// TwinCAT 3 PLC project PlcProject
// ProgramVersion: 3.1.4023.0
// libraries:
//   lcls-twincat-motion, * (SLAC)
//   Tc2_EtherCAT, * (Beckhoff Automation GmbH)
//   Tc2_IoFunctions, * (Beckhoff Automation GmbH)
//   Tc2_MC2, * (Beckhoff Automation GmbH)
//   Tc2_Standard, * (Beckhoff Automation GmbH)
//   Tc2_System, * (Beckhoff Automation GmbH)
//   Tc2_Utilities, * (Beckhoff Automation GmbH)
//   Tc3_Module, * (Beckhoff Automation GmbH)
// project tree:
//   / PlcTask.TcTTO
//   POUs/ MAIN.TcPOU, PRG_VLS_MOTION.TcPOU
// real-time tasks:
//   TASK PlcTask: cycle T#10ms, priority 20, ADS port 350
// motion (NC):
//   TASK NC-Task 1 SAF: cycle T#2ms, priority 4, ADS port 501
//   TASK NC-Task 1 SVB: cycle T#10ms, priority 8, ADS port 511
//   AXIS VLS-Slit-Right (id 1)
//     Dynamic: AccelerationMaximum=10, DecelerationMaximum=10, Acceleration=2.29041, Deceleration=2.29041, Jerk=19.7962
//     Velo: RefSearch=0.1, RefSync=0.1, SlowManual=0.5, FastManual=1, Maximum=0.5
//     OtherSettings: AllowMotionCmdToSlave=true, PulseDistancePos=1, PulseDistanceNeg=1
//     encoder EncType=4
//       EncPara: ScaleFactorNumerator=3.90625e-05, Inverse=true, MaxCount=#x0000ffff
//         SoftEndMinControl: Enable=true, Range=-48.4338
//         SoftEndMaxControl: Enable=true
//         Inc: RefSoftSyncMask=#x0000ffff
//     drive DrvType=24
//       DrvPara: Inverse=true
//         Analog: VeloReferenz=5, ScaleFactorActTorque=0.1
//         TimeComp: TaskDelayCycles=1
//     controller CtrType=2
//       CtrPara: PriorControlFactor=1
//         PosDiffControl: Range=0.1
//         PID: DeadBandPosition=0.1
//         Observer: BandWidth=20
//   AXIS VLS-Slit-Left (id 2)
//     Dynamic: AccelerationMaximum=10, DecelerationMaximum=10, Acceleration=4.49102, Deceleration=4.49102, Jerk=20.1692
//     Velo: RefSearch=0.1, RefSync=0.1, SlowManual=0.5, FastManual=1, Maximum=0.5
//     OtherSettings: AllowMotionCmdToSlave=true, PulseDistancePos=1, PulseDistanceNeg=1
//     encoder EncType=4
//       EncPara: ScaleFactorNumerator=3.90625e-05, MaxCount=#x0000ffff
//         Inc: RefSoftSyncMask=#x0000ffff
//     drive DrvType=24
//       Analog: VeloReferenz=5, ScaleFactorActTorque=0.1
//       TimeComp: TaskDelayCycles=1
//     controller CtrType=2
//       CtrPara: PriorControlFactor=1
//         PosDiffControl: Range=0.1
//         PID: DeadBandPosition=0.1
//         Observer: BandWidth=20
//   AXIS VLS-Slit-Down (id 3)
//     Dynamic: AccelerationMaximum=10, DecelerationMaximum=10, Acceleration=4.49102, Deceleration=4.49102, Jerk=20.1692
//     Velo: RefSearch=0.1, RefSync=0.1, SlowManual=0.5, FastManual=1, Maximum=1
//     OtherSettings: AllowMotionCmdToSlave=true, PulseDistancePos=1, PulseDistanceNeg=1
//     encoder EncType=4
//       EncPara: ScaleFactorNumerator=3.90625e-05, MaxCount=#x0000ffff
//         Inc: RefSoftSyncMask=#x0000ffff
//     drive DrvType=24
//       Analog: VeloReferenz=5, ScaleFactorActTorque=0.1
//       TimeComp: TaskDelayCycles=1
//     controller CtrType=2
//       CtrPara: PriorControlFactor=1
//         PosDiffControl: Range=0.1
//         PID: DeadBandPosition=0.1
//         Observer: BandWidth=20
//   AXIS VLS-Slit-Up (id 4)
//     Dynamic: AccelerationMaximum=10, DecelerationMaximum=10, Acceleration=4.49102, Deceleration=4.49102, Jerk=20.1692
//     Velo: RefSearch=0.1, RefSync=0.1, SlowManual=0.5, FastManual=1, Maximum=1
//     OtherSettings: AllowMotionCmdToSlave=true, PulseDistancePos=1, PulseDistanceNeg=1
//     encoder EncType=4
//       EncPara: ScaleFactorNumerator=3.90625e-05, MaxCount=#x0000ffff
//         Inc: RefSoftSyncMask=#x0000ffff
//     drive DrvType=24
//       Analog: VeloReferenz=5, ScaleFactorActTorque=0.1
//       TimeComp: TaskDelayCycles=1
//     controller CtrType=2
//       CtrPara: PriorControlFactor=1
//         PosDiffControl: Range=0.1
//         PID: DeadBandPosition=0.1
//         Observer: BandWidth=20
//   AXIS VLS-Focus-Mirror (id 5)
//     Dynamic: AccelerationMaximum=4, DecelerationMaximum=4, Acceleration=1.92472, Deceleration=1.92472, Jerk=18.5227
//     Velo: RefSearch=0.05, RefSync=0.05, SlowManual=0.05, FastManual=0.1, Maximum=0.4
//     OtherSettings: AllowMotionCmdToSlave=true, PulseDistancePos=0.1, PulseDistanceNeg=0.1
//     encoder EncType=4
//       EncPara: ScaleFactorNumerator=2.48046875e-05, Inverse=true, MaxCount=#x0000ffff
//         SoftEndMinControl: Enable=true
//         SoftEndMaxControl: Enable=true, Range=4.59
//         Inc: RefSoftSyncMask=#x0000ffff
//     drive DrvType=24
//       DrvPara: Inverse=true
//         Analog: VeloReferenz=3.175, ScaleFactorActTorque=0.1
//         TimeComp: TaskDelayCycles=1
//     controller CtrType=2
//       CtrPara: PriorControlFactor=1
//         PosDiffControl: Range=0.1
//         PID: DeadBandPosition=0.1
//         Observer: BandWidth=20
//   AXIS VLS-Grating (id 6)
//     Dynamic: AccelerationMaximum=10, DecelerationMaximum=10, Acceleration=4.49102, Deceleration=4.49102, Jerk=20.1692
//     Velo: RefSearch=0.1, RefSync=0.1, SlowManual=0.25, FastManual=0.5, Maximum=0.1
//     OtherSettings: AllowMotionCmdToSlave=true, PulseDistancePos=0.5, PulseDistanceNeg=0.5
//     encoder EncType=4
//       EncPara: ScaleFactorNumerator=3.90625e-06, Inverse=true, MaxCount=#x0000ffff
//         SoftEndMinControl: Enable=true
//         SoftEndMaxControl: Enable=true, Range=2.9933
//         Inc: RefSoftSyncMask=#x0000ffff
//     drive DrvType=24
//       DrvPara: Inverse=true
//         Analog: VeloReferenz=0.5, ScaleFactorActTorque=0.1
//         TimeComp: TaskDelayCycles=1
//     controller CtrType=2
//       CtrPara: PriorControlFactor=1
//         PosDiffControl: Range=0.2
//         PID: DeadBandPosition=0.1
//         Observer: BandWidth=20
//   AXIS VLS-Camera-Dist (id 7)
//     Dynamic: AccelerationMaximum=1.8, DecelerationMaximum=1.8, Acceleration=0.89, Deceleration=0.89, Jerk=3.83306
//     Velo: RefSearch=0.05, RefSync=0.05, SlowManual=0.05, FastManual=0.1, Maximum=0.4
//     OtherSettings: AllowMotionCmdToSlave=true, PulseDistancePos=1, PulseDistanceNeg=1
//     encoder EncType=4
//       EncPara: ScaleFactorNumerator=4.097617188e-06, MaxCount=#x0000ffff
//         Inc: RefSoftSyncMask=#x0000ffff
//     drive DrvType=24
//       Analog: VeloReferenz=0.524495, ScaleFactorActTorque=0.1
//       TimeComp: TaskDelayCycles=1
//     controller CtrType=2
//       CtrPara: PriorControlFactor=1
//         PosDiffControl: Range=0.1
//         PID: DeadBandPosition=0.1
//         Observer: BandWidth=20
//   AXIS VLS-Camera-Pitch (id 8)
//     General: UnitName=Degree
//     Dynamic: AccelerationMaximum=0.2, DecelerationMaximum=0.2, Acceleration=0.112494, Deceleration=0.112494, Jerk=0.506199
//     Velo: RefSearch=0.01, RefSync=0.01, SlowManual=0.01, FastManual=0.02, Maximum=0.02
//     OtherSettings: AllowMotionCmdToSlave=true, PulseDistancePos=0.1, PulseDistanceNeg=0.1
//     encoder EncType=4
//       EncPara: ScaleFactorNumerator=5.3515625e-07, Inverse=true, MaxCount=#x0000ffff
//         Inc: RefMode=2, RefSoftSyncMask=#x0000ffff
//     drive DrvType=24
//       DrvPara: Inverse=true
//         Analog: VeloReferenz=0.0685, ScaleFactorActTorque=0.1
//         TimeComp: TaskDelayCycles=1
//     controller CtrType=2
//       CtrPara: PriorControlFactor=1
//         PosDiffControl: Range=0.1
//         PID: DeadBandPosition=0.1
//         Observer: BandWidth=20
// I/O:
//   DEVICE Device 1 (EtherCAT), AmsNetId 5.65.203.216.2.1
//     Term 2 (EK1200) [EK1200-5000 EtherCAT Power supply (2A E-Bus)]
//       Term 1 (EK1122-0008) [EK1122-0008 2 port EtherCAT junction M8]
//         VLS_EP7041-3002_E1 [EP7041-3002 1Ch. Stepper motor output stage (50V, 5A)]
//         VLS_EP7041-3002_E2 [EP7041-3002 1Ch. Stepper motor output stage (50V, 5A)]
//         VLS_EP7041-3002_E3 [EP7041-3002 1Ch. Stepper motor output stage (50V, 5A)]
//         VLS_EP7041-1002_E4 [EP7041-1002 1Ch. Stepper motor output stage (50V, 1.5A)]
//         VLS_EP7041-1002_E5 [EP7041-1002 1Ch. Stepper motor output stage (50V, 1.5A)]
//         VLS_EP7041-1002_E6 [EP7041-1002 1Ch. Stepper motor output stage (50V, 1.5A)]
//         VLS_EP7041-1002_E7 [EP7041-1002 1Ch. Stepper motor output stage (50V, 1.5A)]
//         VLS_EP7041-1002_E8 [EP7041-1002 1Ch. Stepper motor output stage (50V, 1.5A)]
// variable links:
//   (this object) <-> Device 1 (EtherCAT)/Term 2 (EK1200)/Term 1 (EK1122-0008)/VLS_EP7041-3002_E1
//     Drive/Inputs/In/nState1 @bit 3 <-> STM Status/Status/Error
//     Drive/Inputs/In/nState1 @bit 7 <-> STM Status/Status/Motor stall
//     Drive/Inputs/In/nState1 @bit 5 <-> STM Status/Status/Moving negative
//     Drive/Inputs/In/nState1 @bit 4 <-> STM Status/Status/Moving positive
//     Drive/Inputs/In/nState1 @bit 1 <-> STM Status/Status/Ready
//     Drive/Inputs/In/nState1 <-> STM Status/Status/Ready to enable
//     Drive/Inputs/In/nState1 @bit 6 <-> STM Status/Status/Torque reduced
//     Drive/Inputs/In/nState1 @bit 2 <-> STM Status/Status/Warning
//     Drive/Inputs/In/nState2 @bit 3 <-> STM Status/Status/Digital input 1
//     Drive/Inputs/In/nState2 @bit 4 <-> STM Status/Status/Digital input 2
//     Drive/Inputs/In/nState2 @bit 5 <-> STM Status/Status/Sync error
//     Drive/Inputs/In/nState2 @bit 7 <-> STM Status/Status/TxPDO Toggle
//     Drive/Inputs/In/nState4 @bit 1 <-> WcState/InputToggle
//     Drive/Inputs/In/nState4 <-> WcState/WcState
//     Drive/Outputs/Out/nCtrl1 <-> STM Control/Control/Enable
//     Drive/Outputs/Out/nCtrl1 @bit 2 <-> STM Control/Control/Reduce torque
//     Drive/Outputs/Out/nCtrl1 @bit 1 <-> STM Control/Control/Reset
//     Drive/Outputs/Out/nCtrl2 @bit 3 <-> STM Control/Control/Digital output 1
//     Drive/Outputs/Out/nDataOut2[0] <-> STM Velocity/Velocity
//     Enc/Inputs/In/nDataIn1[0] <-> ENC Status compact/Counter value
//     Enc/Inputs/In/nDataIn2[0] <-> ENC Status compact/Latch value
//     Enc/Inputs/In/nState1 @bit 4 <-> ENC Status compact/Status/Counter overflow
//     Enc/Inputs/In/nState1 @bit 3 <-> ENC Status compact/Status/Counter underflow
//     Enc/Inputs/In/nState1 @bit 7 <-> ENC Status compact/Status/Extrapolation stall
//     Enc/Inputs/In/nState1 <-> ENC Status compact/Status/Latch C valid
//     Enc/Inputs/In/nState1 @bit 1 <-> ENC Status compact/Status/Latch extern valid
//     Enc/Inputs/In/nState1 @bit 2 <-> ENC Status compact/Status/Set counter done
//     Enc/Inputs/In/nState2 @bit 4 <-> ENC Status compact/Status/Status of extern latch
//     Enc/Inputs/In/nState2 <-> ENC Status compact/Status/Status of input A
//     Enc/Inputs/In/nState2 @bit 1 <-> ENC Status compact/Status/Status of input B
//     Enc/Inputs/In/nState2 @bit 2 <-> ENC Status compact/Status/Status of input C
//     Enc/Inputs/In/nState2 @bit 5 <-> ENC Status compact/Status/Sync error
//     Enc/Inputs/In/nState2 @bit 7 <-> ENC Status compact/Status/TxPDO Toggle
//     Enc/Inputs/In/nState4 @bit 1 <-> WcState/InputToggle
//     Enc/Inputs/In/nState4 <-> WcState/WcState
//     Enc/Outputs/Out/nCtrl1 <-> ENC Control compact/Control/Enable latch C
//     Enc/Outputs/Out/nCtrl1 @bit 3 <-> ENC Control compact/Control/Enable latch extern on negative edge
//     Enc/Outputs/Out/nCtrl1 @bit 1 <-> ENC Control compact/Control/Enable latch extern on positive edge
//     Enc/Outputs/Out/nCtrl1 @bit 2 <-> ENC Control compact/Control/Set counter
//     Enc/Outputs/Out/nDataOut1[0] <-> ENC Control compact/Set counter value
//   (this object) <-> Device 1 (EtherCAT)/Term 2 (EK1200)/Term 1 (EK1122-0008)/VLS_EP7041-3002_E2
//     Drive/Inputs/In/nState1 @bit 3 <-> STM Status/Status/Error
//     Drive/Inputs/In/nState1 @bit 7 <-> STM Status/Status/Motor stall
//     Drive/Inputs/In/nState1 @bit 5 <-> STM Status/Status/Moving negative
//     Drive/Inputs/In/nState1 @bit 4 <-> STM Status/Status/Moving positive
//     Drive/Inputs/In/nState1 @bit 1 <-> STM Status/Status/Ready
//     Drive/Inputs/In/nState1 <-> STM Status/Status/Ready to enable
//     Drive/Inputs/In/nState1 @bit 6 <-> STM Status/Status/Torque reduced
//     Drive/Inputs/In/nState1 @bit 2 <-> STM Status/Status/Warning
//     Drive/Inputs/In/nState2 @bit 3 <-> STM Status/Status/Digital input 1
//     Drive/Inputs/In/nState2 @bit 4 <-> STM Status/Status/Digital input 2
//     Drive/Inputs/In/nState2 @bit 5 <-> STM Status/Status/Sync error
//     Drive/Inputs/In/nState2 @bit 7 <-> STM Status/Status/TxPDO Toggle
//     Drive/Inputs/In/nState4 @bit 1 <-> WcState/InputToggle
//     Drive/Inputs/In/nState4 <-> WcState/WcState
//     Drive/Outputs/Out/nCtrl1 <-> STM Control/Control/Enable
//     Drive/Outputs/Out/nCtrl1 @bit 2 <-> STM Control/Control/Reduce torque
//     Drive/Outputs/Out/nCtrl1 @bit 1 <-> STM Control/Control/Reset
//     Drive/Outputs/Out/nCtrl2 @bit 3 <-> STM Control/Control/Digital output 1
//     Drive/Outputs/Out/nDataOut2[0] <-> STM Velocity/Velocity
//     Enc/Inputs/In/nDataIn1[0] <-> ENC Status compact/Counter value
//     Enc/Inputs/In/nDataIn2[0] <-> ENC Status compact/Latch value
//     Enc/Inputs/In/nState1 @bit 4 <-> ENC Status compact/Status/Counter overflow
//     Enc/Inputs/In/nState1 @bit 3 <-> ENC Status compact/Status/Counter underflow
//     Enc/Inputs/In/nState1 @bit 7 <-> ENC Status compact/Status/Extrapolation stall
//     Enc/Inputs/In/nState1 <-> ENC Status compact/Status/Latch C valid
//     Enc/Inputs/In/nState1 @bit 1 <-> ENC Status compact/Status/Latch extern valid
//     Enc/Inputs/In/nState1 @bit 2 <-> ENC Status compact/Status/Set counter done
//     Enc/Inputs/In/nState2 @bit 4 <-> ENC Status compact/Status/Status of extern latch
//     Enc/Inputs/In/nState2 <-> ENC Status compact/Status/Status of input A
//     Enc/Inputs/In/nState2 @bit 1 <-> ENC Status compact/Status/Status of input B
//     Enc/Inputs/In/nState2 @bit 2 <-> ENC Status compact/Status/Status of input C
//     Enc/Inputs/In/nState2 @bit 5 <-> ENC Status compact/Status/Sync error
//     Enc/Inputs/In/nState2 @bit 7 <-> ENC Status compact/Status/TxPDO Toggle
//     Enc/Inputs/In/nState4 @bit 1 <-> WcState/InputToggle
//     Enc/Inputs/In/nState4 <-> WcState/WcState
//     Enc/Outputs/Out/nCtrl1 <-> ENC Control compact/Control/Enable latch C
//     Enc/Outputs/Out/nCtrl1 @bit 3 <-> ENC Control compact/Control/Enable latch extern on negative edge
//     Enc/Outputs/Out/nCtrl1 @bit 1 <-> ENC Control compact/Control/Enable latch extern on positive edge
//     Enc/Outputs/Out/nCtrl1 @bit 2 <-> ENC Control compact/Control/Set counter
//     Enc/Outputs/Out/nDataOut1[0] <-> ENC Control compact/Set counter value
//   (this object) <-> Device 1 (EtherCAT)/Term 2 (EK1200)/Term 1 (EK1122-0008)/VLS_EP7041-3002_E3
//     Drive/Inputs/In/nState1 @bit 3 <-> STM Status/Status/Error
//     Drive/Inputs/In/nState1 @bit 7 <-> STM Status/Status/Motor stall
//     Drive/Inputs/In/nState1 @bit 5 <-> STM Status/Status/Moving negative
//     Drive/Inputs/In/nState1 @bit 4 <-> STM Status/Status/Moving positive
//     Drive/Inputs/In/nState1 @bit 1 <-> STM Status/Status/Ready
//     Drive/Inputs/In/nState1 <-> STM Status/Status/Ready to enable
//     Drive/Inputs/In/nState1 @bit 6 <-> STM Status/Status/Torque reduced
//     Drive/Inputs/In/nState1 @bit 2 <-> STM Status/Status/Warning
//     Drive/Inputs/In/nState2 @bit 3 <-> STM Status/Status/Digital input 1
//     Drive/Inputs/In/nState2 @bit 4 <-> STM Status/Status/Digital input 2
//     Drive/Inputs/In/nState2 @bit 5 <-> STM Status/Status/Sync error
//     Drive/Inputs/In/nState2 @bit 7 <-> STM Status/Status/TxPDO Toggle
//     Drive/Inputs/In/nState4 @bit 1 <-> WcState/InputToggle
//     Drive/Inputs/In/nState4 <-> WcState/WcState
//     Drive/Outputs/Out/nCtrl1 <-> STM Control/Control/Enable
//     Drive/Outputs/Out/nCtrl1 @bit 2 <-> STM Control/Control/Reduce torque
//     Drive/Outputs/Out/nCtrl1 @bit 1 <-> STM Control/Control/Reset
//     Drive/Outputs/Out/nCtrl2 @bit 3 <-> STM Control/Control/Digital output 1
//     Drive/Outputs/Out/nDataOut2[0] <-> STM Velocity/Velocity
//     Enc/Inputs/In/nDataIn1[0] <-> ENC Status compact/Counter value
//     Enc/Inputs/In/nDataIn2[0] <-> ENC Status compact/Latch value
//     Enc/Inputs/In/nState1 @bit 4 <-> ENC Status compact/Status/Counter overflow
//     Enc/Inputs/In/nState1 @bit 3 <-> ENC Status compact/Status/Counter underflow
//     Enc/Inputs/In/nState1 @bit 7 <-> ENC Status compact/Status/Extrapolation stall
//     Enc/Inputs/In/nState1 <-> ENC Status compact/Status/Latch C valid
//     Enc/Inputs/In/nState1 @bit 1 <-> ENC Status compact/Status/Latch extern valid
//     Enc/Inputs/In/nState1 @bit 2 <-> ENC Status compact/Status/Set counter done
//     Enc/Inputs/In/nState2 @bit 4 <-> ENC Status compact/Status/Status of extern latch
//     Enc/Inputs/In/nState2 <-> ENC Status compact/Status/Status of input A
//     Enc/Inputs/In/nState2 @bit 1 <-> ENC Status compact/Status/Status of input B
//     Enc/Inputs/In/nState2 @bit 2 <-> ENC Status compact/Status/Status of input C
//     Enc/Inputs/In/nState2 @bit 5 <-> ENC Status compact/Status/Sync error
//     Enc/Inputs/In/nState2 @bit 7 <-> ENC Status compact/Status/TxPDO Toggle
//     Enc/Inputs/In/nState4 @bit 1 <-> WcState/InputToggle
//     Enc/Inputs/In/nState4 <-> WcState/WcState
//     Enc/Outputs/Out/nCtrl1 <-> ENC Control compact/Control/Enable latch C
//     Enc/Outputs/Out/nCtrl1 @bit 3 <-> ENC Control compact/Control/Enable latch extern on negative edge
//     Enc/Outputs/Out/nCtrl1 @bit 1 <-> ENC Control compact/Control/Enable latch extern on positive edge
//     Enc/Outputs/Out/nCtrl1 @bit 2 <-> ENC Control compact/Control/Set counter
//     Enc/Outputs/Out/nDataOut1[0] <-> ENC Control compact/Set counter value
//   (this object) <-> Device 1 (EtherCAT)/Term 2 (EK1200)/Term 1 (EK1122-0008)/VLS_EP7041-1002_E4
//     Drive/Inputs/In/nState1 @bit 3 <-> STM Status/Status/Error
//     Drive/Inputs/In/nState1 @bit 5 <-> STM Status/Status/Moving negative
//     Drive/Inputs/In/nState1 @bit 4 <-> STM Status/Status/Moving positive
//     Drive/Inputs/In/nState1 @bit 1 <-> STM Status/Status/Ready
//     Drive/Inputs/In/nState1 <-> STM Status/Status/Ready to enable
//     Drive/Inputs/In/nState1 @bit 6 <-> STM Status/Status/Torque reduced
//     Drive/Inputs/In/nState1 @bit 2 <-> STM Status/Status/Warning
//     Drive/Inputs/In/nState2 @bit 3 <-> STM Status/Status/Digital input 1
//     Drive/Inputs/In/nState2 @bit 4 <-> STM Status/Status/Digital input 2
//     Drive/Inputs/In/nState2 @bit 5 <-> STM Status/Status/Sync error
//     Drive/Inputs/In/nState2 @bit 7 <-> STM Status/Status/TxPDO Toggle
//     Drive/Inputs/In/nState4 @bit 1 <-> WcState/InputToggle
//     Drive/Inputs/In/nState4 <-> WcState/WcState
//     Drive/Outputs/Out/nCtrl1 <-> STM Control/Control/Enable
//     Drive/Outputs/Out/nCtrl1 @bit 2 <-> STM Control/Control/Reduce torque
//     Drive/Outputs/Out/nCtrl1 @bit 1 <-> STM Control/Control/Reset
//     Drive/Outputs/Out/nCtrl2 @bit 3 <-> STM Control/Control/Digital output 1
//     Drive/Outputs/Out/nDataOut2[0] <-> STM Velocity/Velocity
//     Enc/Inputs/In/nDataIn1[0] <-> ENC Status compact/Counter value
//     Enc/Inputs/In/nDataIn2[0] <-> ENC Status compact/Latch value
//     Enc/Inputs/In/nState1 @bit 4 <-> ENC Status compact/Status/Counter overflow
//     Enc/Inputs/In/nState1 @bit 3 <-> ENC Status compact/Status/Counter underflow
//     Enc/Inputs/In/nState1 @bit 7 <-> ENC Status compact/Status/Extrapolation stall
//     Enc/Inputs/In/nState1 <-> ENC Status compact/Status/Latch C valid
//     Enc/Inputs/In/nState1 @bit 1 <-> ENC Status compact/Status/Latch extern valid
//     Enc/Inputs/In/nState1 @bit 2 <-> ENC Status compact/Status/Set counter done
//     Enc/Inputs/In/nState2 @bit 4 <-> ENC Status compact/Status/Status of extern latch
//     Enc/Inputs/In/nState2 <-> ENC Status compact/Status/Status of input A
//     Enc/Inputs/In/nState2 @bit 1 <-> ENC Status compact/Status/Status of input B
//     Enc/Inputs/In/nState2 @bit 2 <-> ENC Status compact/Status/Status of input C
//     Enc/Inputs/In/nState2 @bit 5 <-> ENC Status compact/Status/Sync error
//     Enc/Inputs/In/nState2 @bit 7 <-> ENC Status compact/Status/TxPDO Toggle
//     Enc/Inputs/In/nState4 @bit 1 <-> WcState/InputToggle
//     Enc/Inputs/In/nState4 <-> WcState/WcState
//     Enc/Outputs/Out/nCtrl1 <-> ENC Control compact/Control/Enable latch C
//     Enc/Outputs/Out/nCtrl1 @bit 3 <-> ENC Control compact/Control/Enable latch extern on negative edge
//     Enc/Outputs/Out/nCtrl1 @bit 1 <-> ENC Control compact/Control/Enable latch extern on positive edge
//     Enc/Outputs/Out/nCtrl1 @bit 2 <-> ENC Control compact/Control/Set counter
//     Enc/Outputs/Out/nDataOut1[0] <-> ENC Control compact/Set counter value
//   (this object) <-> Device 1 (EtherCAT)/Term 2 (EK1200)/Term 1 (EK1122-0008)/VLS_EP7041-1002_E5
//     Drive/Inputs/In/nState1 @bit 3 <-> STM Status/Status/Error
//     Drive/Inputs/In/nState1 @bit 5 <-> STM Status/Status/Moving negative
//     Drive/Inputs/In/nState1 @bit 4 <-> STM Status/Status/Moving positive
//     Drive/Inputs/In/nState1 @bit 1 <-> STM Status/Status/Ready
//     Drive/Inputs/In/nState1 <-> STM Status/Status/Ready to enable
//     Drive/Inputs/In/nState1 @bit 6 <-> STM Status/Status/Torque reduced
//     Drive/Inputs/In/nState1 @bit 2 <-> STM Status/Status/Warning
//     Drive/Inputs/In/nState2 @bit 3 <-> STM Status/Status/Digital input 1
//     Drive/Inputs/In/nState2 @bit 4 <-> STM Status/Status/Digital input 2
//     Drive/Inputs/In/nState2 @bit 5 <-> STM Status/Status/Sync error
//     Drive/Inputs/In/nState2 @bit 7 <-> STM Status/Status/TxPDO Toggle
//     Drive/Inputs/In/nState4 @bit 1 <-> WcState/InputToggle
//     Drive/Inputs/In/nState4 <-> WcState/WcState
//     Drive/Outputs/Out/nCtrl1 <-> STM Control/Control/Enable
//     Drive/Outputs/Out/nCtrl1 @bit 2 <-> STM Control/Control/Reduce torque
//     Drive/Outputs/Out/nCtrl1 @bit 1 <-> STM Control/Control/Reset
//     Drive/Outputs/Out/nCtrl2 @bit 3 <-> STM Control/Control/Digital output 1
//     Drive/Outputs/Out/nDataOut2[0] <-> STM Velocity/Velocity
//     Enc/Inputs/In/nDataIn1[0] <-> ENC Status compact/Counter value
//     Enc/Inputs/In/nDataIn2[0] <-> ENC Status compact/Latch value
//     Enc/Inputs/In/nState1 @bit 4 <-> ENC Status compact/Status/Counter overflow
//     Enc/Inputs/In/nState1 @bit 3 <-> ENC Status compact/Status/Counter underflow
//     Enc/Inputs/In/nState1 @bit 7 <-> ENC Status compact/Status/Extrapolation stall
//     Enc/Inputs/In/nState1 <-> ENC Status compact/Status/Latch C valid
//     Enc/Inputs/In/nState1 @bit 1 <-> ENC Status compact/Status/Latch extern valid
//     Enc/Inputs/In/nState1 @bit 2 <-> ENC Status compact/Status/Set counter done
//     Enc/Inputs/In/nState2 @bit 4 <-> ENC Status compact/Status/Status of extern latch
//     Enc/Inputs/In/nState2 <-> ENC Status compact/Status/Status of input A
//     Enc/Inputs/In/nState2 @bit 1 <-> ENC Status compact/Status/Status of input B
//     Enc/Inputs/In/nState2 @bit 2 <-> ENC Status compact/Status/Status of input C
//     Enc/Inputs/In/nState2 @bit 5 <-> ENC Status compact/Status/Sync error
//     Enc/Inputs/In/nState2 @bit 7 <-> ENC Status compact/Status/TxPDO Toggle
//     Enc/Inputs/In/nState4 @bit 1 <-> WcState/InputToggle
//     Enc/Inputs/In/nState4 <-> WcState/WcState
//     Enc/Outputs/Out/nCtrl1 <-> ENC Control compact/Control/Enable latch C
//     Enc/Outputs/Out/nCtrl1 @bit 3 <-> ENC Control compact/Control/Enable latch extern on negative edge
//     Enc/Outputs/Out/nCtrl1 @bit 1 <-> ENC Control compact/Control/Enable latch extern on positive edge
//     Enc/Outputs/Out/nCtrl1 @bit 2 <-> ENC Control compact/Control/Set counter
//     Enc/Outputs/Out/nDataOut1[0] <-> ENC Control compact/Set counter value
//   (this object) <-> Device 1 (EtherCAT)/Term 2 (EK1200)/Term 1 (EK1122-0008)/VLS_EP7041-1002_E6
//     Drive/Inputs/In/nState1 @bit 3 <-> STM Status/Status/Error
//     Drive/Inputs/In/nState1 @bit 5 <-> STM Status/Status/Moving negative
//     Drive/Inputs/In/nState1 @bit 4 <-> STM Status/Status/Moving positive
//     Drive/Inputs/In/nState1 @bit 1 <-> STM Status/Status/Ready
//     Drive/Inputs/In/nState1 <-> STM Status/Status/Ready to enable
//     Drive/Inputs/In/nState1 @bit 6 <-> STM Status/Status/Torque reduced
//     Drive/Inputs/In/nState1 @bit 2 <-> STM Status/Status/Warning
//     Drive/Inputs/In/nState2 @bit 3 <-> STM Status/Status/Digital input 1
//     Drive/Inputs/In/nState2 @bit 4 <-> STM Status/Status/Digital input 2
//     Drive/Inputs/In/nState2 @bit 5 <-> STM Status/Status/Sync error
//     Drive/Inputs/In/nState2 @bit 7 <-> STM Status/Status/TxPDO Toggle
//     Drive/Inputs/In/nState4 @bit 1 <-> WcState/InputToggle
//     Drive/Inputs/In/nState4 <-> WcState/WcState
//     Drive/Outputs/Out/nCtrl1 <-> STM Control/Control/Enable
//     Drive/Outputs/Out/nCtrl1 @bit 2 <-> STM Control/Control/Reduce torque
//     Drive/Outputs/Out/nCtrl1 @bit 1 <-> STM Control/Control/Reset
//     Drive/Outputs/Out/nCtrl2 @bit 3 <-> STM Control/Control/Digital output 1
//     Drive/Outputs/Out/nDataOut2[0] <-> STM Velocity/Velocity
//     Enc/Inputs/In/nDataIn1[0] <-> ENC Status compact/Counter value
//     Enc/Inputs/In/nDataIn2[0] <-> ENC Status compact/Latch value
//     Enc/Inputs/In/nState1 @bit 4 <-> ENC Status compact/Status/Counter overflow
//     Enc/Inputs/In/nState1 @bit 3 <-> ENC Status compact/Status/Counter underflow
//     Enc/Inputs/In/nState1 @bit 7 <-> ENC Status compact/Status/Extrapolation stall
//     Enc/Inputs/In/nState1 <-> ENC Status compact/Status/Latch C valid
//     Enc/Inputs/In/nState1 @bit 1 <-> ENC Status compact/Status/Latch extern valid
//     Enc/Inputs/In/nState1 @bit 2 <-> ENC Status compact/Status/Set counter done
//     Enc/Inputs/In/nState2 @bit 4 <-> ENC Status compact/Status/Status of extern latch
//     Enc/Inputs/In/nState2 <-> ENC Status compact/Status/Status of input A
//     Enc/Inputs/In/nState2 @bit 1 <-> ENC Status compact/Status/Status of input B
//     Enc/Inputs/In/nState2 @bit 2 <-> ENC Status compact/Status/Status of input C
//     Enc/Inputs/In/nState2 @bit 5 <-> ENC Status compact/Status/Sync error
//     Enc/Inputs/In/nState2 @bit 7 <-> ENC Status compact/Status/TxPDO Toggle
//     Enc/Inputs/In/nState4 @bit 1 <-> WcState/InputToggle
//     Enc/Inputs/In/nState4 <-> WcState/WcState
//     Enc/Outputs/Out/nCtrl1 <-> ENC Control compact/Control/Enable latch C
//     Enc/Outputs/Out/nCtrl1 @bit 3 <-> ENC Control compact/Control/Enable latch extern on negative edge
//     Enc/Outputs/Out/nCtrl1 @bit 1 <-> ENC Control compact/Control/Enable latch extern on positive edge
//     Enc/Outputs/Out/nCtrl1 @bit 2 <-> ENC Control compact/Control/Set counter
//     Enc/Outputs/Out/nDataOut1[0] <-> ENC Control compact/Set counter value
//   (this object) <-> Device 1 (EtherCAT)/Term 2 (EK1200)/Term 1 (EK1122-0008)/VLS_EP7041-1002_E7
//     Drive/Inputs/In/nState1 @bit 3 <-> STM Status/Status/Error
//     Drive/Inputs/In/nState1 @bit 5 <-> STM Status/Status/Moving negative
//     Drive/Inputs/In/nState1 @bit 4 <-> STM Status/Status/Moving positive
//     Drive/Inputs/In/nState1 @bit 1 <-> STM Status/Status/Ready
//     Drive/Inputs/In/nState1 <-> STM Status/Status/Ready to enable
//     Drive/Inputs/In/nState1 @bit 6 <-> STM Status/Status/Torque reduced
//     Drive/Inputs/In/nState1 @bit 2 <-> STM Status/Status/Warning
//     Drive/Inputs/In/nState2 @bit 3 <-> STM Status/Status/Digital input 1
//     Drive/Inputs/In/nState2 @bit 4 <-> STM Status/Status/Digital input 2
//     Drive/Inputs/In/nState2 @bit 5 <-> STM Status/Status/Sync error
//     Drive/Inputs/In/nState2 @bit 7 <-> STM Status/Status/TxPDO Toggle
//     Drive/Inputs/In/nState4 @bit 1 <-> WcState/InputToggle
//     Drive/Inputs/In/nState4 <-> WcState/WcState
//     Drive/Outputs/Out/nCtrl1 <-> STM Control/Control/Enable
//     Drive/Outputs/Out/nCtrl1 @bit 2 <-> STM Control/Control/Reduce torque
//     Drive/Outputs/Out/nCtrl1 @bit 1 <-> STM Control/Control/Reset
//     Drive/Outputs/Out/nCtrl2 @bit 3 <-> STM Control/Control/Digital output 1
//     Drive/Outputs/Out/nDataOut2[0] <-> STM Velocity/Velocity
//     Enc/Inputs/In/nDataIn1[0] <-> ENC Status compact/Counter value
//     Enc/Inputs/In/nDataIn2[0] <-> ENC Status compact/Latch value
//     Enc/Inputs/In/nState1 @bit 4 <-> ENC Status compact/Status/Counter overflow
//     Enc/Inputs/In/nState1 @bit 3 <-> ENC Status compact/Status/Counter underflow
//     Enc/Inputs/In/nState1 @bit 7 <-> ENC Status compact/Status/Extrapolation stall
//     Enc/Inputs/In/nState1 <-> ENC Status compact/Status/Latch C valid
//     Enc/Inputs/In/nState1 @bit 1 <-> ENC Status compact/Status/Latch extern valid
//     Enc/Inputs/In/nState1 @bit 2 <-> ENC Status compact/Status/Set counter done
//     Enc/Inputs/In/nState2 @bit 4 <-> ENC Status compact/Status/Status of extern latch
//     Enc/Inputs/In/nState2 <-> ENC Status compact/Status/Status of input A
//     Enc/Inputs/In/nState2 @bit 1 <-> ENC Status compact/Status/Status of input B
//     Enc/Inputs/In/nState2 @bit 2 <-> ENC Status compact/Status/Status of input C
//     Enc/Inputs/In/nState2 @bit 5 <-> ENC Status compact/Status/Sync error
//     Enc/Inputs/In/nState2 @bit 7 <-> ENC Status compact/Status/TxPDO Toggle
//     Enc/Inputs/In/nState4 @bit 1 <-> WcState/InputToggle
//     Enc/Inputs/In/nState4 <-> WcState/WcState
//     Enc/Outputs/Out/nCtrl1 <-> ENC Control compact/Control/Enable latch C
//     Enc/Outputs/Out/nCtrl1 @bit 3 <-> ENC Control compact/Control/Enable latch extern on negative edge
//     Enc/Outputs/Out/nCtrl1 @bit 1 <-> ENC Control compact/Control/Enable latch extern on positive edge
//     Enc/Outputs/Out/nCtrl1 @bit 2 <-> ENC Control compact/Control/Set counter
//     Enc/Outputs/Out/nDataOut1[0] <-> ENC Control compact/Set counter value
//   (this object) <-> Device 1 (EtherCAT)/Term 2 (EK1200)/Term 1 (EK1122-0008)/VLS_EP7041-1002_E8
//     Drive/Inputs/In/nState1 @bit 3 <-> STM Status/Status/Error
//     Drive/Inputs/In/nState1 @bit 5 <-> STM Status/Status/Moving negative
//     Drive/Inputs/In/nState1 @bit 4 <-> STM Status/Status/Moving positive
//     Drive/Inputs/In/nState1 @bit 1 <-> STM Status/Status/Ready
//     Drive/Inputs/In/nState1 <-> STM Status/Status/Ready to enable
//     Drive/Inputs/In/nState1 @bit 6 <-> STM Status/Status/Torque reduced
//     Drive/Inputs/In/nState1 @bit 2 <-> STM Status/Status/Warning
//     Drive/Inputs/In/nState2 @bit 3 <-> STM Status/Status/Digital input 1
//     Drive/Inputs/In/nState2 @bit 4 <-> STM Status/Status/Digital input 2
//     Drive/Inputs/In/nState2 @bit 5 <-> STM Status/Status/Sync error
//     Drive/Inputs/In/nState2 @bit 7 <-> STM Status/Status/TxPDO Toggle
//     Drive/Inputs/In/nState4 @bit 1 <-> WcState/InputToggle
//     Drive/Inputs/In/nState4 <-> WcState/WcState
//     Drive/Outputs/Out/nCtrl1 <-> STM Control/Control/Enable
//     Drive/Outputs/Out/nCtrl1 @bit 2 <-> STM Control/Control/Reduce torque
//     Drive/Outputs/Out/nCtrl1 @bit 1 <-> STM Control/Control/Reset
//     Drive/Outputs/Out/nCtrl2 @bit 3 <-> STM Control/Control/Digital output 1
//     Drive/Outputs/Out/nDataOut2[0] <-> STM Velocity/Velocity
//     Enc/Inputs/In/nDataIn1[0] <-> ENC Status compact/Counter value
//     Enc/Inputs/In/nDataIn2[0] <-> ENC Status compact/Latch value
//     Enc/Inputs/In/nState1 @bit 4 <-> ENC Status compact/Status/Counter overflow
//     Enc/Inputs/In/nState1 @bit 3 <-> ENC Status compact/Status/Counter underflow
//     Enc/Inputs/In/nState1 @bit 7 <-> ENC Status compact/Status/Extrapolation stall
//     Enc/Inputs/In/nState1 <-> ENC Status compact/Status/Latch C valid
//     Enc/Inputs/In/nState1 @bit 1 <-> ENC Status compact/Status/Latch extern valid
//     Enc/Inputs/In/nState1 @bit 2 <-> ENC Status compact/Status/Set counter done
//     Enc/Inputs/In/nState2 @bit 4 <-> ENC Status compact/Status/Status of extern latch
//     Enc/Inputs/In/nState2 <-> ENC Status compact/Status/Status of input A
//     Enc/Inputs/In/nState2 @bit 1 <-> ENC Status compact/Status/Status of input B
//     Enc/Inputs/In/nState2 @bit 2 <-> ENC Status compact/Status/Status of input C
//     Enc/Inputs/In/nState2 @bit 5 <-> ENC Status compact/Status/Sync error
//     Enc/Inputs/In/nState2 @bit 7 <-> ENC Status compact/Status/TxPDO Toggle
//     Enc/Inputs/In/nState4 @bit 1 <-> WcState/InputToggle
//     Enc/Inputs/In/nState4 <-> WcState/WcState
//     Enc/Outputs/Out/nCtrl1 <-> ENC Control compact/Control/Enable latch C
//     Enc/Outputs/Out/nCtrl1 @bit 3 <-> ENC Control compact/Control/Enable latch extern on negative edge
//     Enc/Outputs/Out/nCtrl1 @bit 1 <-> ENC Control compact/Control/Enable latch extern on positive edge
//     Enc/Outputs/Out/nCtrl1 @bit 2 <-> ENC Control compact/Control/Set counter
//     Enc/Outputs/Out/nDataOut1[0] <-> ENC Control compact/Set counter value
//   vls_motion Instance <-> Device 1 (EtherCAT)/Term 2 (EK1200)/Term 1 (EK1122-0008)/VLS_EP7041-1002_E4
//     PlcTask Inputs/Main.M4.bLimitBackwardEnable <-> STM Status/Status/Digital input 1
//     PlcTask Inputs/Main.M4.bLimitForwardEnable <-> STM Status/Status/Digital input 2
//   vls_motion Instance <-> Device 1 (EtherCAT)/Term 2 (EK1200)/Term 1 (EK1122-0008)/VLS_EP7041-1002_E5
//     PlcTask Inputs/Main.M5.bLimitBackwardEnable <-> STM Status/Status/Digital input 2
//     PlcTask Inputs/Main.M5.bLimitForwardEnable <-> STM Status/Status/Digital input 1
//   vls_motion Instance <-> Device 1 (EtherCAT)/Term 2 (EK1200)/Term 1 (EK1122-0008)/VLS_EP7041-1002_E6
//     PlcTask Inputs/Main.M6.bLimitBackwardEnable <-> STM Status/Status/Digital input 2
//     PlcTask Inputs/Main.M6.bLimitForwardEnable <-> STM Status/Status/Digital input 1
//   vls_motion Instance <-> Device 1 (EtherCAT)/Term 2 (EK1200)/Term 1 (EK1122-0008)/VLS_EP7041-1002_E7
//     PlcTask Inputs/Main.M7.bLimitBackwardEnable <-> STM Status/Status/Digital input 2
//     PlcTask Inputs/Main.M7.bLimitForwardEnable <-> STM Status/Status/Digital input 1
//   vls_motion Instance <-> Device 1 (EtherCAT)/Term 2 (EK1200)/Term 1 (EK1122-0008)/VLS_EP7041-1002_E8
//     PlcTask Inputs/Main.M8.bLimitBackwardEnable <-> STM Status/Status/Digital input 2
//     PlcTask Inputs/Main.M8.bLimitForwardEnable <-> STM Status/Status/Digital input 1
//   vls_motion Instance <-> Device 1 (EtherCAT)/Term 2 (EK1200)/Term 1 (EK1122-0008)/VLS_EP7041-3002_E1
//     PlcTask Inputs/Main.M1.bLimitBackwardEnable <-> STM Status/Status/Digital input 1
//     PlcTask Inputs/Main.M1.bLimitForwardEnable <-> STM Status/Status/Digital input 2
//   vls_motion Instance <-> Device 1 (EtherCAT)/Term 2 (EK1200)/Term 1 (EK1122-0008)/VLS_EP7041-3002_E2
//     PlcTask Inputs/Main.M2.bLimitBackwardEnable <-> STM Status/Status/Digital input 1
//     PlcTask Inputs/Main.M2.bLimitForwardEnable <-> STM Status/Status/Digital input 2
//   vls_motion Instance <-> Device 1 (EtherCAT)/Term 2 (EK1200)/Term 1 (EK1122-0008)/VLS_EP7041-3002_E3
//     PlcTask Inputs/Main.M3.bLimitBackwardEnable <-> STM Status/Status/Digital input 2
//     PlcTask Inputs/Main.M3.bLimitForwardEnable <-> STM Status/Status/Digital input 1
//   vls_motion Instance <-> NC-Task 1 SAF/Axes/VLS-Camera-Dist
//     PlcTask Inputs/Main.M7.Axis.NcToPlc <-> Outputs/ToPlc
//     PlcTask Outputs/Main.M7.Axis.PlcToNc <-> Inputs/FromPlc
//   vls_motion Instance <-> NC-Task 1 SAF/Axes/VLS-Camera-Pitch
//     PlcTask Inputs/Main.M8.Axis.NcToPlc <-> Outputs/ToPlc
//     PlcTask Outputs/Main.M8.Axis.PlcToNc <-> Inputs/FromPlc
//   vls_motion Instance <-> NC-Task 1 SAF/Axes/VLS-Focus-Mirror
//     PlcTask Inputs/Main.M5.Axis.NcToPlc <-> Outputs/ToPlc
//     PlcTask Outputs/Main.M5.Axis.PlcToNc <-> Inputs/FromPlc
//   vls_motion Instance <-> NC-Task 1 SAF/Axes/VLS-Grating
//     PlcTask Inputs/Main.M6.Axis.NcToPlc <-> Outputs/ToPlc
//     PlcTask Outputs/Main.M6.Axis.PlcToNc <-> Inputs/FromPlc
//   vls_motion Instance <-> NC-Task 1 SAF/Axes/VLS-Slit-Down
//     PlcTask Inputs/Main.M3.Axis.NcToPlc <-> Outputs/ToPlc
//     PlcTask Outputs/Main.M3.Axis.PlcToNc <-> Inputs/FromPlc
//   vls_motion Instance <-> NC-Task 1 SAF/Axes/VLS-Slit-Left
//     PlcTask Inputs/Main.M2.Axis.NcToPlc <-> Outputs/ToPlc
//     PlcTask Outputs/Main.M2.Axis.PlcToNc <-> Inputs/FromPlc
//   vls_motion Instance <-> NC-Task 1 SAF/Axes/VLS-Slit-Right
//     PlcTask Inputs/Main.M1.Axis.NcToPlc <-> Outputs/ToPlc
//     PlcTask Outputs/Main.M1.Axis.PlcToNc <-> Inputs/FromPlc
//   vls_motion Instance <-> NC-Task 1 SAF/Axes/VLS-Slit-Up
//     PlcTask Inputs/Main.M4.Axis.NcToPlc <-> Outputs/ToPlc
//     PlcTask Outputs/Main.M4.Axis.PlcToNc <-> Inputs/FromPlc

CONFIGURATION PlcProject
    RESOURCE PLC ON TwinCAT3
        TASK PlcTask(INTERVAL := T#10ms, PRIORITY := 20);
        PROGRAM MAIN WITH PlcTask : MAIN;
    END_RESOURCE
END_CONFIGURATION

// ---- POUs/MAIN.TcPOU
PROGRAM MAIN
VAR

END_VAR

PRG_VLS_MOTION(); // So, run the program associated with coupler

END_PROGRAM

// ---- POUs/PRG_VLS_MOTION.TcPOU
PROGRAM PRG_VLS_MOTION
VAR
	 // VLS Motor 1; VLS-Slit-Right
	{attribute 'TcLinkTo' := '	.bLimitForwardEnable:=TIIB[VLS_EP7041-3002_E1]^STM Status^Status^Digital input 1;
								.bLimitBackwardEnable:=TIIB[VLS_EP7041-3002_E1]^STM Status^Status^Digital input 2'}
    {attribute 'pytmc' := '
        pv: TMO:VLS:MMS:SR
        field: DESC VLS Right Slit Blade
    '}
    M1: DUT_MotionStage;
    fbMotion1: FB_MotionStage;

	 // VLS Motor 2; VLS-Slit-Left
	{attribute 'TcLinkTo' := '	.bLimitForwardEnable:=TIIB[VLS_EP7041-3002_E2]^STM Status^Status^Digital input 1;
								.bLimitBackwardEnable:=TIIB[VLS_EP7041-3002_E2]^STM Status^Status^Digital input 2'}
    {attribute 'pytmc' := '
        pv: TMO:VLS:MMS:SL
        field: DESC VLS Left Slit Blade
    '}
    M2: DUT_MotionStage;
    fbMotion2: FB_MotionStage;
	
	// VLS Motor 3; VLS-Slit-Down
	{attribute 'TcLinkTo' := '	.bLimitForwardEnable:=TIIB[VLS_EP7041-3002_E3]^STM Status^Status^Digital input 1;
								.bLimitBackwardEnable:=TIIB[VLS_EP7041-3002_E3]^STM Status^Status^Digital input 2'}
    {attribute 'pytmc' := '
        pv: TMO:VLS:MMS:SD
        field: DESC VLS Lower Slit Blade
    '}
    M3: DUT_MotionStage;
    fbMotion3: FB_MotionStage;
	
	
	// VLS Motor 4; VLS-Slit-Up
	{attribute 'TcLinkTo' := '	.bLimitForwardEnable:=TIIB[VLS_EP7041-1002_E4]^STM Status^Status^Digital input 1;
								.bLimitBackwardEnable:=TIIB[VLS_EP7041-1002_E4]^STM Status^Status^Digital input 2'}
    {attribute 'pytmc' := '
        pv: pv: TMO:VLS:MMS:SU
        field: DESC VLS Upper Slit Blade
    '}
    M4: DUT_MotionStage;
    fbMotion4: FB_MotionStage;
	
	
	
	// VLS Motor 5; focusing mirror
	{attribute 'TcLinkTo' := '	.bLimitForwardEnable:=TIIB[VLS_EP7041-1002_E5]^STM Status^Status^Digital input 1;
								.bLimitBackwardEnable:=TIIB[VLS_EP7041-1002_E5]^STM Status^Status^Digital input 2'}
    {attribute 'pytmc' := '
        pv: TMO:VLS:MMS:FM
        field: DESC VLS Focus Mirror
    '}
    M5: DUT_MotionStage;
    fbMotion5: FB_MotionStage;
	
	// VLS Motor 6; grating
	{attribute 'TcLinkTo' := '	.bLimitForwardEnable:=TIIB[VLS_EP7041-1002_E6]^STM Status^Status^Digital input 1;
								.bLimitBackwardEnable:=TIIB[VLS_EP7041-1002_E6]^STM Status^Status^Digital input 2'}
    {attribute 'pytmc' := '
        pv: TMO:VLS:MMS:GP
        field: DESC VLS Grating
    '}
    M6: DUT_MotionStage;
    fbMotion6: FB_MotionStage;
	
	// VLS Motor 7; camera translation
	{attribute 'TcLinkTo' := '	.bLimitForwardEnable:=TIIB[VLS_EP7041-1002_E7]^STM Status^Status^Digital input 1;
								.bLimitBackwardEnable:=TIIB[VLS_EP7041-1002_E7]^STM Status^Status^Digital input 2'}
    {attribute 'pytmc' := '
        pv: TMO:VLS:MMS:CD
        field: DESC VLS Camera Distance
    '}
    M7: DUT_MotionStage;
    fbMotion7: FB_MotionStage;
	
	// VLS Motor 8; camera pitch
	{attribute 'TcLinkTo' := '	.bLimitForwardEnable:=TIIB[VLS_EP7041-1002_E8]^STM Status^Status^Digital input 1;
								.bLimitBackwardEnable:=TIIB[VLS_EP7041-1002_E8]^STM Status^Status^Digital input 2'}
    {attribute 'pytmc' := '
        pv: TMO:VLS:MMS:CP
        field: DESC VLS Camera Pitch
    '}
    M8: DUT_MotionStage;
    fbMotion8: FB_MotionStage;

	
	//persistent data
	fbWritePersistentData	: WritePersistentData;
	bInit					: BOOL := TRUE;
	fbWriteDelay			: TON;
	mcSetPosition			: ARRAY [1..8] of MC_SetPosition;
END_VAR

VAR PERSISTENT
	fSlitRightPos	: LREAL;
	fSlitLeftPos	: LREAL;
	fSlitDownPos	: LREAL;
	fSlitUpPos		: LREAL;
	fFocusMirrorPos	: LREAL;
	fGratingPos		: LREAL;
	fCameraDistPos	: LREAL;
	fCameraPitchPos	: LREAL;

END_VAR

IF bInit THEN
	//Sets axes position with persistent value
	mcSetPosition[1](Axis:=M1.Axis, Position:=fSlitRightPos, Mode:=FALSE, Execute:=TRUE);
	mcSetPosition[2](Axis:=M2.Axis, Position:=fSlitLeftPos, Mode:=FALSE, Execute:=TRUE);
	mcSetPosition[3](Axis:=M3.Axis, Position:=fSlitDownPos, Mode:=FALSE, Execute:=TRUE);
	mcSetPosition[4](Axis:=M4.Axis, Position:=fSlitUpPos, Mode:=FALSE, Execute:=TRUE);
	mcSetPosition[5](Axis:=M5.Axis, Position:=fFocusMirrorPos, Mode:=FALSE, Execute:=TRUE);
	mcSetPosition[6](Axis:=M6.Axis, Position:=fGratingPos, Mode:=FALSE, Execute:=TRUE);
	mcSetPosition[7](Axis:=M7.Axis, Position:=fCameraDistPos, Mode:=FALSE, Execute:=TRUE);
	mcSetPosition[8](Axis:=M8.Axis, Position:=fCameraPitchPos, Mode:=FALSE, Execute:=TRUE);
	if (mcSetPosition[1].Done AND mcSetPosition[2].Done AND mcSetPosition[3].Done AND mcSetPosition[4].Done AND 
	mcSetPosition[5].Done AND mcSetPosition[6].Done AND mcSetPosition[7].Done AND mcSetPosition[8].Done) THEN
		bInit:=FALSE;
		mcSetPosition[1](Axis:=M1.Axis, Execute:=FALSE);
		mcSetPosition[2](Axis:=M2.Axis, Execute:=FALSE);
		mcSetPosition[3](Axis:=M3.Axis, Execute:=FALSE);
		mcSetPosition[4](Axis:=M4.Axis, Execute:=FALSE);
		mcSetPosition[5](Axis:=M5.Axis, Execute:=FALSE);
		mcSetPosition[6](Axis:=M6.Axis, Execute:=FALSE);
		mcSetPosition[7](Axis:=M7.Axis, Execute:=FALSE);
		mcSetPosition[8](Axis:=M8.Axis, Execute:=FALSE);
	END_IF
ELSE
	
	M1.nEnableMode := Enum_StageEnableMode.ALWAYS;
	M1.bHardwareEnable := TRUE;
	M1.bPowerSelf := TRUE;
	//M1.bLimitForwardEnable := (M1.bLimitForwardEnable AND M1.bLimitBackwardEnable);
	//M1.bLimitBackwardEnable := (M1.bLimitForwardEnable AND M1.bLimitBackwardEnable);
	fbMotion1(stMotionStage := M1); // top slit blade
	
	M2.nEnableMode := Enum_StageEnableMode.ALWAYS;
	M2.bHardwareEnable := TRUE;
	M2.bPowerSelf := TRUE;
	//M2.bLimitForwardEnable := (M2.bLimitForwardEnable AND M2.bLimitBackwardEnable);
	//M2.bLimitBackwardEnable := (M2.bLimitForwardEnable AND M2.bLimitBackwardEnable);
	fbMotion2(stMotionStage := M2); // bottom slit blade
	
	M3.nEnableMode := Enum_StageEnableMode.ALWAYS;
	M3.bHardwareEnable := TRUE;
	M3.bPowerSelf := TRUE;
	//M3.bLimitForwardEnable := (M3.bLimitForwardEnable AND M3.bLimitBackwardEnable);
	//M3.bLimitBackwardEnable := (M3.bLimitForwardEnable AND M3.bLimitBackwardEnable);
	fbMotion3(stMotionStage := M3); // right slit blade
	
	M4.nEnableMode := Enum_StageEnableMode.ALWAYS;
	M4.bHardwareEnable := TRUE;
	M4.bPowerSelf := TRUE;
	//M4.bLimitForwardEnable := (M4.bLimitForwardEnable AND M4.bLimitBackwardEnable);
	//M4.bLimitBackwardEnable := (M4.bLimitForwardEnable AND M4.bLimitBackwardEnable);
	fbMotion4(stMotionStage := M4); // left slit blade
	
	M5.nEnableMode := Enum_StageEnableMode.ALWAYS;
	M5.bHardwareEnable := TRUE;
	M5.bPowerSelf := TRUE;
	//M5.bLimitForwardEnable := (M5.bLimitForwardEnable AND M5.bLimitBackwardEnable);
	//M5.bLimitBackwardEnable := (M5.bLimitForwardEnable AND M5.bLimitBackwardEnable);
	fbMotion5(stMotionStage := M5); // focusing mirror
	
	M6.nEnableMode := Enum_StageEnableMode.ALWAYS;
	M6.bHardwareEnable := TRUE;
	M6.bPowerSelf := TRUE;
	//M6.bLimitForwardEnable := (M6.bLimitForwardEnable AND M6.bLimitBackwardEnable);
	//M6.bLimitBackwardEnable := (M6.bLimitForwardEnable AND M6.bLimitBackwardEnable);
	fbMotion6(stMotionStage := M6); // grating
	
	M7.nEnableMode := Enum_StageEnableMode.ALWAYS;
	M7.bHardwareEnable := TRUE;
	M7.bPowerSelf := TRUE;
	//M7.bLimitForwardEnable := (M7.bLimitForwardEnable AND M7.bLimitBackwardEnable);
	//M7.bLimitBackwardEnable := (M7.bLimitForwardEnable AND M7.bLimitBackwardEnable);
	fbMotion7(stMotionStage := M7); // camera pitch
	
	M8.nEnableMode := Enum_StageEnableMode.ALWAYS;
	M8.bHardwareEnable := TRUE;
	M8.bPowerSelf := TRUE;
	//M8.bLimitForwardEnable := (M8.bLimitForwardEnable AND M8.bLimitBackwardEnable);
	//M8.bLimitBackwardEnable := (M8.bLimitForwardEnable AND M8.bLimitBackwardEnable);
	fbMotion8(stMotionStage := M8); // camera translation

	
	//Keep track of positions
	fSlitRightPos	:= M1.Axis.NcToPlc.ActPos;
	fSlitLeftPos	:= M2.Axis.NcToPlc.ActPos;
	fSlitDownPos	:= M3.Axis.NcToPlc.ActPos;
	fSlitUpPos		:= M4.Axis.NcToPlc.ActPos;
	fFocusMirrorPos	:= M5.Axis.NcToPlc.ActPos;
	fGratingPos		:= M6.Axis.NcToPlc.ActPos;
	fCameraDistPos	:= M7.Axis.NcToPlc.ActPos;
	fCameraPitchPos	:= M8.Axis.NcToPlc.ActPos;
END_IF

END_PROGRAM
